{attribute addProperty BoxType "EL3783-0000-0018"}
{attribute addProperty Id "I2_SamplesAT %I*ARRAY [0..19] OF INT32040"}
{attribute addProperty CRC "806776176"}
{attribute addProperty SizeInBites "320"}
{attribute addProperty SizeInBytes "40"}
TYPE L2_Current_Samples_30166D70 :
STRUCT
	{attribute addProperty Name "I2_Samples"}
	I2_Samples AT %I* : ARRAY [0..19] OF INT;
END_STRUCT
END_TYPE

(* stored: Version 1.2.0.0, ProductVersion 3.1.4024.9
   DUT L2_Current_Samples_30166D70: Id {0dc91aa3-b709-473b-a2f0-0e7a3361c5ba} *)
